PROGRAM PRG_ALARMS
VAR
	fbTimer			: TON ; 			//
	fbDateTime		: FB_DATE_TIME;		//
	fbAlarmManager	: FB_ALARM_MANAGER;	//

	_Date : STRING;		//DATA IN STRING FORMAT
	_Time : STRING;		//HOUR IN STRING FORMAT
	
(* Variaveis de exemplo para acionamento dos alarmes *)	
	Condition_01: BOOL;	//TEST TO SIMULATE ALARM 1
	Condition_02: BOOL;	//TEST TO SIMULATE ALARM 2
	Condition_03: BOOL;	//TEST TO SIMULATE EVENT 1
	Condition_04: BOOL;	//TEST TO SIMULATE EVENT 2	
END_VAR

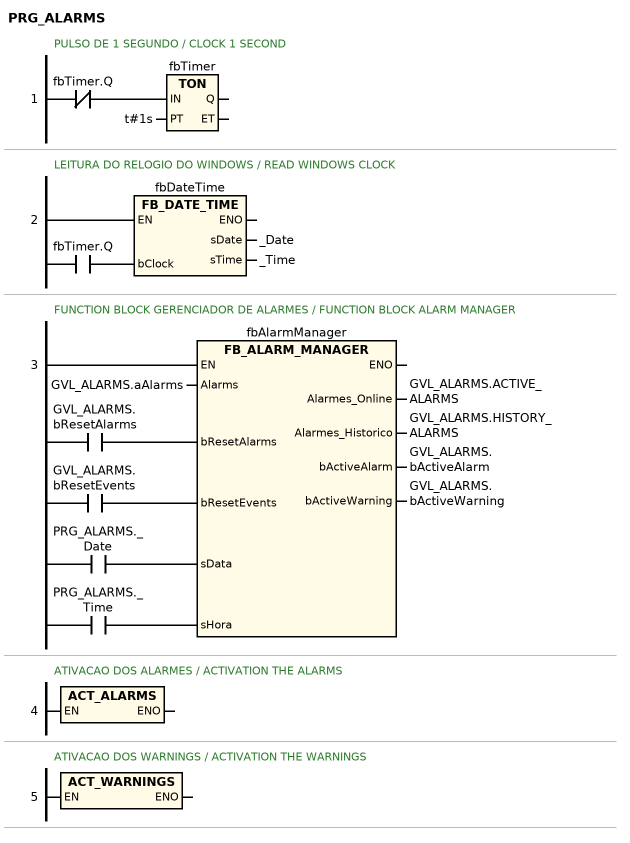
// NETWORK 1
// PULSO DE 1 SEGUNDO / CLOCK 1 SECOND
fbTimer(IN := NOT fbTimer.Q, PT := t#1s); // TON

// NETWORK 2
// LEITURA DO RELOGIO DO WINDOWS / READ WINDOWS CLOCK
fbDateTime(bClock := fbTimer.Q, sDate => _Date, sTime => _Time); // FB_DATE_TIME

// NETWORK 3
// FUNCTION BLOCK GERENCIADOR DE ALARMES / FUNCTION BLOCK ALARM MANAGER
fbAlarmManager(
    Alarms := GVL_ALARMS.aAlarms,
    bResetAlarms := GVL_ALARMS.bResetAlarms,
    bResetEvents := GVL_ALARMS.bResetEvents,
    sData := PRG_ALARMS._Date,
    sHora := PRG_ALARMS._Time,
    Alarmes_Online => GVL_ALARMS.ACTIVE_ALARMS,
    Alarmes_Historico => GVL_ALARMS.HISTORY_ALARMS,
    bActiveAlarm => GVL_ALARMS.bActiveAlarm,
    bActiveWarning => GVL_ALARMS.bActiveWarning); // FB_ALARM_MANAGER

// NETWORK 4
// ATIVACAO DOS ALARMES / ACTIVATION THE ALARMS
ACT_ALARMS();

// NETWORK 5
// ATIVACAO DOS WARNINGS / ACTIVATION THE WARNINGS
ACT_WARNINGS();

ACTION ACT_ALARMS:
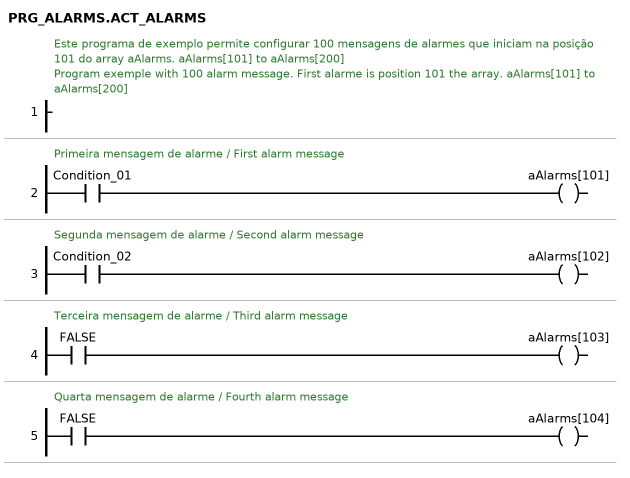
// NETWORK 1
// Este programa de exemplo permite configurar 100 mensagens de alarmes que iniciam na posição 101 do array aAlarms. aAlarms[101] to aAlarms[200]
// Program exemple with 100 alarm message. First alarme is position 101 the array. aAlarms[101] to aAlarms[200]

// NETWORK 2
// Primeira mensagem de alarme / First alarm message
aAlarms[101] := Condition_01;

// NETWORK 3
// Segunda mensagem de alarme / Second alarm message
aAlarms[102] := Condition_02;

// NETWORK 4
// Terceira mensagem de alarme / Third alarm message
aAlarms[103] := FALSE;

// NETWORK 5
// Quarta mensagem de alarme / Fourth alarm message
aAlarms[104] := FALSE;
END_ACTION

ACTION ACT_WARNINGS:
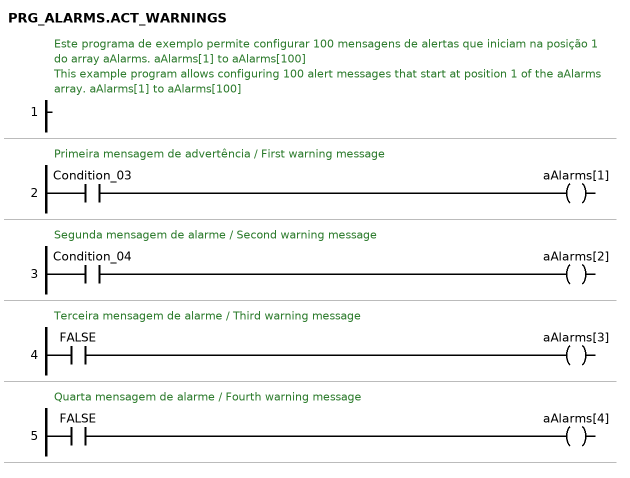
// NETWORK 1
// Este programa de exemplo permite configurar 100 mensagens de alertas que iniciam na posição 1 do array aAlarms. aAlarms[1] to aAlarms[100]
// This example program allows configuring 100 alert messages that start at position 1 of the aAlarms array. aAlarms[1] to aAlarms[100]

// NETWORK 2
// Primeira mensagem de advertência / First warning message
aAlarms[1] := Condition_03;

// NETWORK 3
// Segunda mensagem de alarme / Second warning message
aAlarms[2] := Condition_04;

// NETWORK 4
// Terceira mensagem de alarme / Third warning message
aAlarms[3] := FALSE;

// NETWORK 5
// Quarta mensagem de alarme / Fourth warning message
aAlarms[4] := FALSE;
END_ACTION

END_PROGRAM

(* stored: Version 1.1.0.1, ProductVersion 3.1.4024.12
   POU PRG_ALARMS: Id {81c562e6-b38f-45a0-8afc-79af5f0a0a27}, SpecialFunc None
   Action ACT_ALARMS: Id {2b12135f-85b4-4bdb-828a-337ed0d24145}
   Action ACT_WARNINGS: Id {2c7f7091-4c19-47c4-86ae-ccdeec81e1bb} *)
